# EPICS substitutions: epics/db/EL7201.substitutions
file "./db/ecSlave.template"
{
  pattern {}
          {}
}

file "./db/EL7201.template"
{
  pattern {}
          {}
}
